// TIA Portal V16 export
// export: Created 2024-09-05T17:39:19.5896161Z, ExportSetting WithDefaults, DisplayName Totally Integrated Automation Portal, DisplayVersion V16 Update 6, DisplayName TIA Portal Version Control Interface, DisplayVersion V16 Update 2, DisplayName TIA Portal Openness, DisplayVersion V16 Update 6, DisplayName STEP 7 Professional, DisplayVersion V16 Update 6, DisplayName STEP 7 Safety, DisplayVersion V16, DisplayName WinCC Advanced, DisplayVersion V16 Update 6
DATA_BLOCK "HMIMain_DB"   // DB49
VERSION : 0.1
// stored: AutoNumber true, DBAccessibleFromOPCUA true, InstanceOfName HMIMain, InstanceOfType FB
"HMIMain"
   // VAR
   //    res : Bool := FALSE;
   // END_VAR
BEGIN
END_DATA_BLOCK
